{attribute 'qualified_only'}
VAR_GLOBAL
	mb_Input_Registers   :ARRAY[0..20] OF INT;	// Modbus Adress 32768 Funciton Code 04
END_VAR

(* stored: Version 1.1.0.1, ProductVersion 3.1.4024.11
   GVL GVL: Id {e39b5210-68e1-4653-a13a-6f35dfffebe2} *)
